FUNCTION_BLOCK PUBLIC EcMasterFrameStats IMPLEMENTS IEcTask
VAR_INPUT
END_VAR
VAR_OUTPUT
END_VAR
VAR
	iState : INT;
	masterFrameStats : Tc2_EtherCAT.FB_EcMasterFrameStatistic;
	_execute: BOOL;
	_done: BOOL;
	_busy: BOOL;
	_error: BOOL;
	_netId: AMSNETID;
END_VAR

CASE iState OF
	0:
		IF _execute THEN
			_done := FALSE;
			_busy := TRUE;
			_error := FALSE;
			masterFrameStats.bExecute := TRUE;
			IF masterFrameStats.bBusy THEN
				iState := 10;
				_execute := false;
			END_IF
		END_IF
	10:
		IF NOT masterFrameStats.bBusy THEN
			IF NOT masterFrameStats.bError THEN
				_done := TRUE;
			ELSE
				_error := TRUE;
			END_IF
			_busy := FALSE;
			masterFrameStats.bExecute := FALSE;
			iState := 0;
		END_IF
END_CASE

masterFrameStats(sNetId := Tc2_System.F_CreateAmsNetId(nIds := NetId));

{warning 'add method implementation '}
METHOD Abort : BOOL
masterFrameStats.bExecute := FALSE;
_busy := FALSE;
_execute := FALSE;
Abort := TRUE;
iState := 0;
END_METHOD

{warning 'add property implementation'}
PROPERTY Busy : BOOL
GET
Busy := _busy;
END_GET
END_PROPERTY

{warning 'add property implementation'}
PROPERTY Done : BOOL
GET
Done := _done;
END_GET
END_PROPERTY

{warning 'add property implementation'}
PROPERTY Error : BOOL
GET
Error := _error;
END_GET
END_PROPERTY

METHOD Execute : BOOL
VAR_INPUT
END_VAR
IF NOT Busy THEN
	Execute := _execute := TRUE;
END_IF
END_METHOD

PROPERTY FramesPerSecond  : LREAL
GET
FramesPerSecond := masterFrameStats.fFramesPerSecond;
END_GET
END_PROPERTY

PROPERTY LostFrames : UDINT
GET
LostFrames := masterFrameStats.nLostFrames;
END_GET
END_PROPERTY

PROPERTY LostQueuedFrames : udint
GET
LostQueuedFrames := masterFrameStats.nLostQueuedFrames;
END_GET
END_PROPERTY

{warning 'add property implementation'}
PROPERTY NetID : amsnetid
GET
NetID := _netId;
END_GET
SET
_netId := NetID;
END_SET
END_PROPERTY

PROPERTY QueuedFramesPerSecond : lreal
GET
QueuedFramesPerSecond := masterFrameStats.fQueuedFramesPerSecond;
END_GET
END_PROPERTY

END_FUNCTION_BLOCK

(* stored: Version 1.1.0.1, ProductVersion 3.1.4024.11
   POU EcMasterFrameStats: Id {0413a492-8e64-4a8a-a602-dee5af2e7896}, SpecialFunc None
   Method Abort: Id {93e82a1b-6970-422b-b061-d279b2418e13}
   Property Busy: Id {10d2f24b-9c28-41bc-894d-d0b8e9ef37e5}
   Get Get: Id {2f26ef72-7b44-426c-b562-e959b69a3eb1}
   Property Done: Id {bebea6d1-e9c9-47c8-ab57-d40d151a4baf}
   Get Get: Id {16805e6c-b47e-45ec-b102-e48311973c40}
   Property Error: Id {fca1a19f-f3f0-4440-8c41-51c9edc1ae54}
   Get Get: Id {c7d76716-e4c4-425a-aa7c-2c92059db891}
   Method Execute: Id {40b5d161-faf6-48fb-ba4d-510273399f62}
   Property FramesPerSecond: Id {6e6fa49c-94c2-49bf-8bdb-2d4a74fd5434}
   Get Get: Id {b47865fa-e1a5-4aeb-9d35-beef7507107a}
   Property LostFrames: Id {50dc00be-18e5-49f3-96fd-c664a3c7bd87}
   Get Get: Id {aad2e118-8637-4a9b-b166-c49e0f8d4019}
   Property LostQueuedFrames: Id {dc88780d-37fd-465d-8ee3-84041e07fa1b}
   Get Get: Id {f2974af3-15ca-4fa9-a0d9-620aaccda86c}
   Property NetID: Id {9d7b148c-f32e-4da2-b023-b7f7246c6899}
   Get Get: Id {09335829-c871-4023-b9a5-7fd879876958}
   Set Set: Id {1800f40b-dc45-40c3-a014-03ba4a20f672}
   Property QueuedFramesPerSecond: Id {eaf89791-c3c1-40c0-8944-01ed5c2d6b24}
   Get Get: Id {14444e4d-7775-4073-a411-ce96dbf3fb70} *)
